FUNCTION_BLOCK FB_LoggerTests EXTENDS FB_TestSuite
VAR_INPUT
END_VAR
VAR_OUTPUT
END_VAR
VAR
	fbLogger		: FB_Logger;
	fbFileHandler	: FB_FileHandler;
END_VAR

Test_LogError();
Test_LogWarning();
Test_LogInfo();
Test_LogGeneric();

METHOD Test_LogError
VAR_INPUT
END_VAR

VAR_INST
	bWrite	: BOOL := TRUE;
	TonMaxDelayForFileToAppear	: TON := (PT :=T#2s);
END_VAR
TcUnit.TEST('Test_LogError');

fbLogger.FileProperties.FileLocation := 'C:\';
fbLogger.FileProperties.FileName := 'TestLog';
IF bWrite THEN
	fbLogger.LogError('Error text....');
	bWrite := FALSE;
END_IF

TonMaxDelayForFileToAppear(IN := TRUE);
IF TonMaxDelayForFileToAppear.Q THEN
;
END_IF

fbLogger();


fbFileHandler.FileProperties := fbLogger.FileProperties;
END_METHOD

METHOD Test_LogGeneric
VAR_INPUT
END_VAR
END_METHOD

METHOD Test_LogInfo
VAR_INPUT
END_VAR
END_METHOD

METHOD Test_LogWarning
VAR_INPUT
END_VAR
END_METHOD

END_FUNCTION_BLOCK

(* stored: Version 1.1.0.1, ProductVersion 3.1.4024.13
   POU FB_LoggerTests: Id {56576e73-0b8d-04b4-2a1d-ddaf5d4df6a5}, SpecialFunc None
   Method Test_LogError: Id {d8907491-afae-0e50-10f7-6c16a49476f3}
   Method Test_LogGeneric: Id {85c6ce0a-a15b-043a-2e4c-eb245e65cfdf}
   Method Test_LogInfo: Id {36be4fe7-4f92-0086-3d7c-e81a29d0db62}
   Method Test_LogWarning: Id {4fe293bd-ef31-0f9e-0f9c-a610eddd16dc} *)
